{attribute addProperty BoxType "EJ3048-0000-0020"}
{attribute addProperty Id "StatusAT %I*Status_F0C7FE3C1621ValueAT %I*INT16217"}
{attribute addProperty CRC "4050261517"}
{attribute addProperty SizeInBites "32"}
{attribute addProperty SizeInBytes "4"}
TYPE AI_Standard_Channel_F16A160D :
STRUCT
	{attribute addProperty Name "Status"}
	Status AT %I* : Status_F0C7FE3C;
	{attribute addProperty Name "Value"}
	Value AT %I* : INT;
END_STRUCT
END_TYPE

(* stored: Version 1.2.0.0, ProductVersion 3.1.4024.9
   DUT AI_Standard_Channel_F16A160D: Id {074b453f-9532-4d8c-b115-1bda9be73f5f} *)
